INTERFACE O_Sensor

PROPERTY isTriggered : BOOL
GET
END_GET
END_PROPERTY

END_INTERFACE

(* stored: Version 1.1.0.1, ProductVersion 3.1.4024.12
   Itf O_Sensor: Id {1bb325d0-1cfe-4fee-8786-696ebce98699}
   Property isTriggered: Id {6eeb55dd-f52f-4836-a1f2-b796588547c0}
   Get Get: Id {33fe77af-4230-4f6d-8b1f-93cae4f77eea} *)
